Universal Robots PolyScope program: TTS_BAM_-675_700.urp

Program TTS_BAM_-675_700 (installation=default directory=/programs/Benoit/Maria createdIn=5.24.0 lastSavedIn=5.24.0 robotSerialNumber=20256701031)
Calibrated DH parameters: a=[0.000298, -0.647434, -0.453269, 0.000079, -0.000017, 0]; d=[0.218696, -1.643942, -72.520022, 74.346318, 0.136008, 0.143459]; alpha=[1.571299, 0.009127, 0.003331, 1.569882, -1.570435, 0]; deltaTheta=[-0.000001, -0.02317, 5.807334, 0.499029, 0.000006, 0]
InitVariablesNode
Robot Program (runOnlyOnce=true)
  SafeHome (positionOptionType=SPEED_AND_ACCELERATION speed=1.047198 acceleration=1.396263 nextMotionTime=2)
  MoveJ speed 60 deg/s, acceleration 80 deg/s^2 (useActiveTCP=true optimoveEnabled=false optiMoveSpeed=0.2 optiMoveAcceleration=0.04) feature=Base
    Waypoint Waypoint_2: TCP in base x=-199.99 y=-400 z=799.996 mm, rx=0 ry=0 rz=1.5708 rad; joints [-92.945, -173.316, 128.949, 134.384, -89.566, -266.771] deg
  MoveL speed 250 mm/s, acceleration 1200 mm/s^2 (useActiveTCP=true optimoveEnabled=false optiMoveSpeed=0.2 optiMoveAcceleration=0.04) feature=Base
    Waypoint Waypoint_1: TCP in base x=-999.99 y=-675 z=700 mm, rx=0 ry=0 rz=1.5708 rad; joints [-137.428, -178.107, 35.593, 232.533, -89.32, -222.485] deg; TCP offset x=0 y=0 z=0 mm, rx=0 ry=0 rz=0 rad
  SuppressedNode
    Script file /programs/TTS_BAM/force_approach.script
      | # -------------------------------------------------
      | # Force approach in Tool Z+
      | # Max travel: 100 mm
      | # If target force is reached: hold for 2 seconds
      | # Then return to exact starting pose
      | # -------------------------------------------------
      | 
      | # USER SETTINGS
      | target_force = 250.0
      | force_reached_limit = 230.0
      | 
      | max_travel = 0.120          # 100 mm
      | hold_time_cycles = 250      # approx. 2 seconds at 125 Hz
      | 
      | force_speed_limit = 0.05   # 10 mm/s
      | 
      | return_acc = 0.05
      | return_speed = 0.1
      | 
      | 
      | # -------------------------------------------------
      | # Save exact current pose before starting
      | # -------------------------------------------------
      | 
      | return_pose = get_actual_tcp_pose()
      | 
      | # We also use this same pose as the force reference frame.
      | force_start_pose = return_pose
      | 
      | 
      | # -------------------------------------------------
      | # Prepare force mode
      | # -------------------------------------------------
      | 
      | zero_ftsensor()
      | 
      | task_frame = force_start_pose
      | selection_vector = [0, 0, 1, 0, 0, 0]
      | wrench = [0, 0, target_force, 0, 0, 0]
      | force_type = 2
      | 
      | # For compliant Z, third value is the speed limit in m/s.
      | limits = [0.1, 0.1, force_speed_limit, 0.17, 0.17, 0.17]
      | 
      | force_reached = False
      | travel_limit_reached = False
      | 
      | 
      | # -------------------------------------------------
      | # Approach phase
      | # Stop when force is reached OR 100 mm travel is reached
      | # -------------------------------------------------
      | 
      | while force_reached == False and travel_limit_reached == False:
      | 
      |   force_mode(task_frame, selection_vector, wrench, force_type, limits)
      | 
      |   current_pose = get_actual_tcp_pose()
      | 
      |   # Current TCP pose relative to starting TCP pose
      |   relative_pose = pose_trans(pose_inv(force_start_pose), current_pose)
      | 
      |   # Travel along original Tool Z+
      |   z_travel = relative_pose[2]
      | 
      |   current_force = force()
      | 
      |   if current_force >= force_reached_limit:
      |     force_reached = True
      |   end
      | 
      |   if z_travel >= max_travel:
      |     travel_limit_reached = True
      |   end
      | 
      |   sync()
      | 
      | end
      | 
      | 
      | # -------------------------------------------------
      | # Hold phase
      | # Only hold if the force was actually reached
      | # -------------------------------------------------
      | 
      | if force_reached == True:
      | 
      |   hold_count = 0
      | 
      |   while hold_count < hold_time_cycles:
      | 
      |     force_mode(task_frame, selection_vector, wrench, force_type, limits)
      | 
      |     hold_count = hold_count + 1
      | 
      |     sync()
      | 
      |   end
      | 
      | end
      | 
      | 
      | # -------------------------------------------------
      | # End force mode and return to exact starting pose
      | # -------------------------------------------------
      | 
      | end_force_mode()
      | 
      | # Stop any remaining force-mode movement smoothly
      | stopl(0.5)
      | 
      | if force_reached == True:
      | sleep(2.0)
      | end
      | 
      | 
      | # Return to the exact TCP pose from before the force approach
      | movel(return_pose, a=return_acc, v=return_speed, r=0)
  Loop Counting (count=10) loopVariable(name=Loop_1)
    Script file /programs/TTS_BAM/force_approach.script
      | (same text as the earlier copy of this file)
    MoveL speed 250 mm/s, acceleration 1200 mm/s^2 (useActiveTCP=true optimoveEnabled=false optiMoveSpeed=0.2 optiMoveAcceleration=0.04) feature=Base
      MoveDirectionNode (selectedDirection=XPlus)
        Until DISTANCE (allowActions=false deceleration=3 distanceNodeType=STOP) Distance=0.2; motionParameters(blendRadius=0)
  Script file /programs/TTS_BAM/force_approach.script
    | (same text as the earlier copy of this file)
  MoveJ speed 60 deg/s, acceleration 80 deg/s^2 (useActiveTCP=true optimoveEnabled=false optiMoveSpeed=0.2 optiMoveAcceleration=0.04) feature=Base
    Waypoint Waypoint_2: TCP in base x=-199.99 y=-400 z=799.996 mm, rx=0 ry=0 rz=1.5708 rad; joints [-92.945, -173.316, 128.949, 134.384, -89.566, -266.771] deg
